INTERFACE I_XTS_Station_PLC EXTENDS I_CH_Object

METHOD ChangePos : HRESULT
VAR_INPUT
	fNewPosOnTrack : LREAL;
END_VAR
END_METHOD

(*The _ PLC interface provides the user with a simplified interface for commanding between the stations. Sometimes, however, this is not enough. 
Either you get the corresponding interface with the __Queryinterface or you can get full access with this property.*)
PROPERTY FullAccess : I_XTS_Station
GET
END_GET
END_PROPERTY

{attribute 'monitoring':='call'}
PROPERTY LUID : STRING
GET
END_GET
END_PROPERTY

{attribute 'monitoring':='call'}
PROPERTY MoverQueueSize : UINT
GET
END_GET
SET
END_SET
END_PROPERTY

{attribute 'monitoring':='call'}
PROPERTY MoversInPlace : BOOL
GET
END_GET
END_PROPERTY

{attribute 'monitoring':='call'}
PROPERTY MoversInQueue : REFERENCE TO ARRAY [0..(XtsParameterlist.MAX_MOVER_PER_SYSTEM-1)] OF I_XTS_Mover_PLC // Return a sorted list of movers in this zone. Index 0 is the mover in Front.
GET
END_GET
END_PROPERTY

{attribute 'monitoring':='call'}
PROPERTY MoverVelocityAtExit : LREAL //[mm/s] Every mover that leaves or passes the station gets this new velocity as a target.
GET
END_GET
SET
END_SET
END_PROPERTY

{attribute 'monitoring':='call'}
PROPERTY PositionOnTrack : LREAL
GET
END_GET
END_PROPERTY

{attribute 'monitoring':='call'}
PROPERTY ProcessSimulationActive : BOOL
GET
END_GET
END_PROPERTY

{attribute 'monitoring':='call'}
//prevent further movers from entering the station, 
//e.g. to prevent a collision. All movers that are already moving to reach this station will be stopped with a stop 
//and restarted with Ready True.
PROPERTY ReadyToRecvMovers : BOOL
GET
END_GET
SET
END_SET
END_PROPERTY

METHOD SendMoversToStation : HRESULT
VAR_INPUT
	sTargedStation : STRING;
END_VAR
END_METHOD

//If a valid time (>0seconds) is set and the configured destination station exists, then the movers will be sent away automatically after this time from now on.
METHOD SimulationStart : HRESULT
VAR_INPUT
	fProcessDuration 	: LREAL; //[s]
	sTargedStation		: STRING; //LUID of the targed station to automatic send after the duration
END_VAR
END_METHOD

//If a valid time (>0seconds) is set and the configured destination station exists, then the movers will be sent away automatically after this time from now on.
METHOD SimulationStartEx : HRESULT
VAR_INPUT
	fProcessDuration 		: LREAL; //[s]
	ipStation				: I_Xts_Station_PLC; //unique station to automatic send after the duration
END_VAR
END_METHOD

METHOD SimulationStop : HRESULT
END_METHOD

{attribute 'monitoring':='call'}
PROPERTY SuppressDynamicsChange : BOOL
GET
END_GET
SET
END_SET
END_PROPERTY

{attribute 'monitoring':='call'}
//A time that is waited as soon as the mover is in the station (including the monitoring window) before “MoversInPlace” is set. e.g. used to stabilize the workpiece
PROPERTY TargetPosMonitoringTime : TIME
GET
END_GET
SET
END_SET
END_PROPERTY

{attribute 'monitoring':='call'}
//How many mm before the mover reaches the position is “MoversInPlace” set for the process. 
//This distance can also be set very large (e.g. 100mm) for moving past without stopping.
PROPERTY TargetPosWindow : LREAL
GET
END_GET
SET
END_SET
END_PROPERTY

END_INTERFACE

(* stored: Version 1.1.0.1, ProductVersion 3.1.4024.12
   Itf I_XTS_Station_PLC: Id {daddfa80-c9fa-4c49-900c-a6fb951bb190}
   Folder Simulation: Id {789658cf-b705-40c0-94f0-535859f81ba3}
   Method ChangePos: Id {8f1bbf6f-89e4-46fa-b5f9-5fd8a664821c}
   Property FullAccess: Id {45e62743-3387-478b-9a60-985dc203b931}
   Get Get: Id {61c8deea-134e-4df0-8bd7-1c4b66b48426}
   Property LUID: Id {f51ef214-629a-4fbd-a29d-a1e604692fad}
   Get Get: Id {ed3877a4-c9d3-42f9-9ffd-ef20ae1f50b6}
   Property MoverQueueSize: Id {e6a5c534-744e-40c7-9a6d-d0395bc146a5}
   Get Get: Id {6a0f7267-66fb-43c2-8a16-dbfba4eb4512}
   Set Set: Id {46965e05-dc77-4ac1-82ec-964c5b28f9be}
   Property MoversInPlace: Id {d140a936-d829-49d6-b510-6e1536fc5359}
   Get Get: Id {7d5cf4eb-009d-4b41-8186-3dfeb57b0212}
   Property MoversInQueue: Id {bfdaff81-6320-4707-9ee0-4fc7d9e27b60}
   Get Get: Id {bfd8e5b5-9dd9-4b9e-bfa4-82fa0fc4a9ef}
   Property MoverVelocityAtExit: Id {f2944c40-39e9-4526-a477-ab0d4da33829}
   Get Get: Id {d2dce039-d70a-4e7e-abc5-5079a4396125}
   Set Set: Id {55c83297-a46f-4fae-a9ad-25b99775423e}
   Property PositionOnTrack: Id {895a03a0-b6dd-44ba-9c3d-0b0fc2c8cace}
   Get Get: Id {dfb11930-293d-4ada-810b-2fd784122e2f}
   Property ProcessSimulationActive: Id {1b022c27-2795-4ab7-8f8b-c212d8182f66}
   Get Get: Id {838ef149-d373-4e9f-a5cb-23dd6ca61950}
   Property ReadyToRecvMovers: Id {48f1dc5e-dcf0-4f66-8110-6c04e80873c8}
   Get Get: Id {95091e33-bd4c-4a50-85f5-0492ab9d9f3d}
   Set Set: Id {9f534000-9dd0-4710-93f4-5efd056ac4d8}
   Method SendMoversToStation: Id {9ffcc3ee-c8e5-4481-8022-b7e502b12478}
   Method SimulationStart: Id {4455c854-ccc4-4c79-8b12-75eea6adf457}
   Method SimulationStartEx: Id {335c4ff8-afb5-4d3d-9388-94804580560f}
   Method SimulationStop: Id {e562dd1e-1297-41c0-8396-bdd0d555dfec}
   Property SuppressDynamicsChange: Id {8dd724d4-7d4b-4ca2-a807-764f9e122ee0}
   Get Get: Id {f4ee8745-fc48-4fc5-ba64-1f3047bb4d14}
   Set Set: Id {698940c6-031f-4343-b689-6b9e6e2fa94b}
   Property TargetPosMonitoringTime: Id {8424cad3-fafb-429e-9a48-80b6febb946d}
   Get Get: Id {b356251f-51a7-4e5d-b49b-5c8e96965fca}
   Set Set: Id {711c14cf-2709-4fcf-81e6-bfa70f785a21}
   Property TargetPosWindow: Id {7278d6f6-3c30-4905-8b4f-d7802dfba026}
   Get Get: Id {5ae39e46-8d6c-4690-b782-2e57cbaa6746}
   Set Set: Id {36589e9d-82c1-4d40-a94c-36f20fc410b3} *)
